{attribute 'qualified_only'}
VAR_GLOBAL
	newTrunks:BOOL;
	dddj:int;
END_VAR

(* stored: Version 1.1.0.1, ProductVersion 3.1.4022.17
   GVL GVL: Id {de70d6a0-78c3-4872-9217-9dd6f1616ebb} *)
